TYPE ST_TcpVisionOutImm :
STRUCT
    LinkState    : E_ByteChannelState;
    LastResponse : STRING(255);
END_STRUCT
END_TYPE

(* stored: Version 1.1.0.1, ProductVersion 3.1.4024.12
   DUT ST_TcpVisionOutImm: Id {e3668539-4981-4891-ae2e-9c18d31e5854} *)
